TYPE ST_TxRx :
STRUCT
	sSend : STRING;
	sReceived: STRING;
END_STRUCT
END_TYPE

(* stored: Version 1.1.0.1, ProductVersion 3.1.4020.6
   DUT ST_TxRx: Id {5aac0779-84bd-411e-abd2-8d4fed6dcd03} *)
